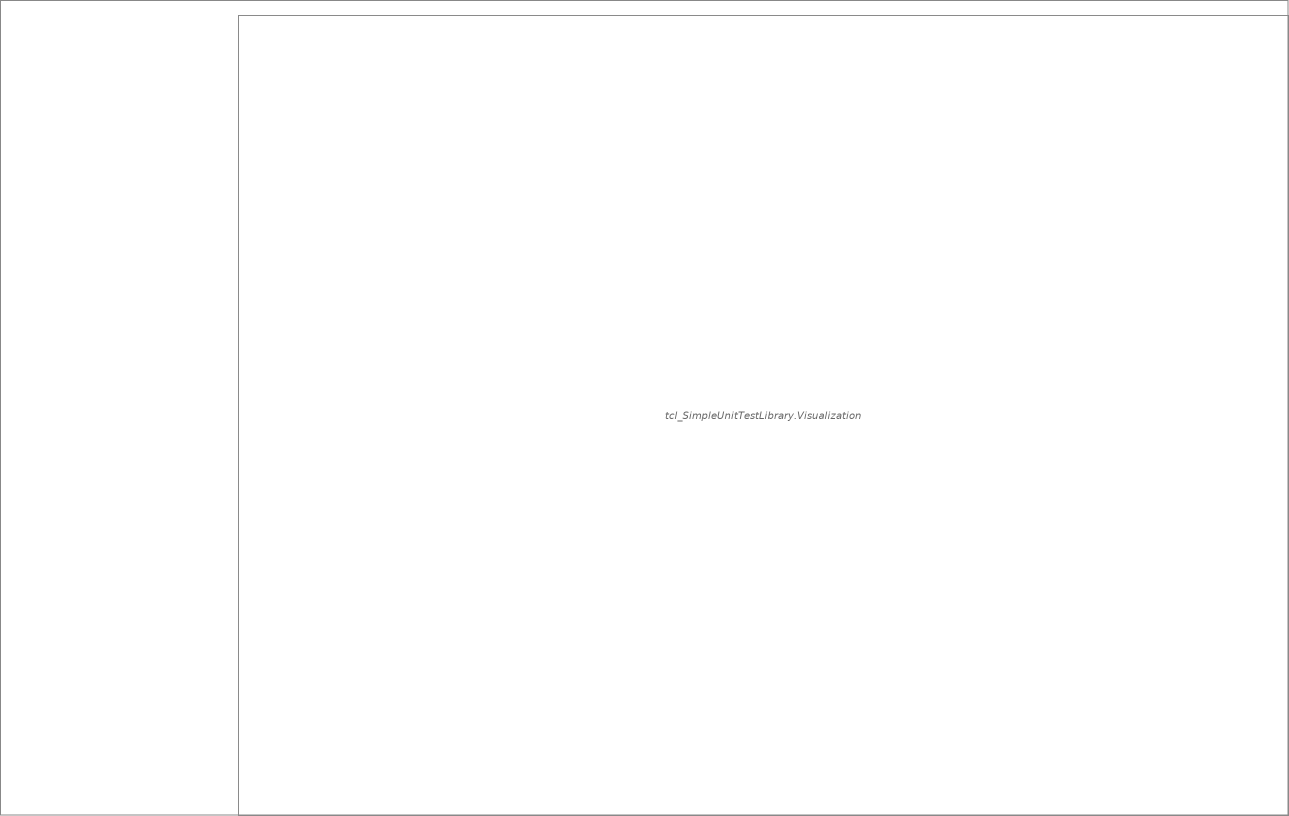
VISUALIZATION TestUI  // 1289x816
    Frame (238,15 1051x801)
        shows tcl_SimpleUnitTestLibrary.Visualization(TestRunner := MAIN.testRunner)
END_VISUALIZATION

(* stored: Version 1.1.0.1, ProductVersion 3.1.4024.13
   Visu TestUI: Id {663724fa-6b1f-45fc-8640-b1279cbc7657} *)
